{attribute 'qualified_only'}
{attribute 'strict'}
TYPE E_PosTest :
(
	Idle_start :=0,
	GoToNextState_levelHi := 1,
	GoToNextState_levelLo := 2,
	MovingTo_levelHi :=3,
	MovingTo_levelLo :=4,
	Idle_init :=5
);
END_TYPE

(* stored: Version 1.1.0.1, ProductVersion 3.1.4024.6
   DUT E_PosTest: Id {3fe16123-87a5-4b15-9302-05b0cfbb18fc} *)
